FUNCTION F_Leerfahren : BOOL
VAR_INPUT
END_VAR
VAR
END_VAR

(* Netzwerk: 3 Leerfahren *)

(*
	O "M8.1MagLeerf" M8.1 -- Magazin Leerfahren
	O "M8.2SortLeerf" M8.2 -- Sortierer Leerfahren
	S "M 23.1" M23.1 -- Zylinder sollen IN Leerfahrstellung
*)	
IF VAT.bMagazinLeerfahren OR VAT.bSortiererLeerfahren THEN
	VAT.bZylINLeerFahrt := TRUE; //Zylinder sollen IN Leerfahrstellung
END_IF

(*	
	UN "M8.1MagLeerf" M8.1 -- Magazin Leerfahren
	UN "M8.2SortLeerf" M8.2 -- Sortierer Leerfahren
	U "M 23.1" M23.1 -- Zylinder sollen IN Leerfahrstellung
	R "M 23.1" M23.1 -- Zylinder sollen IN Leerfahrstellung
	S "M 23.2" M23.2 -- Zylinder sollen AUS Leerfahrstellung
*)
IF NOT VAT.bMagazinLeerfahren AND
	NOT VAT.bSortiererLeerfahren AND
	VAT.bZylINLeerFahrt THEN
	
	VAT.bZylINLeerFahrt := FALSE;
	VAT.bZylAUSLeerFahrt := TRUE;
END_IF

(*	
	O "M 23.0" M23.0 -- Takt für Vereinzelung bei Leerfahren
	SPBN kl
*)

IF NOT VAT.bTaktVereinzLeerF THEN
	RETURN;
END_IF

(*	
	U "T 41" T41 -- Takt für Magazin leerfahren
	SPB kl
*)
GVL.tofMagazLeerFahr(IN := FALSE, PT := T#500MS);
IF GVL.tofMagazLeerFahr.Q THEN
	RETURN;
END_IF

(*
	L S5T#500MS
	SA "T 41" T41 -- Takt für Magazin leerfahren
	CLR
	SA "T 41" T41 -- Takt für Magazin leerfahren
	
	UN "M 23.0" M23.0 -- Takt für Vereinzelung bei Leerfahren
	= "M 23.0" M23.0 -- Takt für Vereinzelung bei Leerfahren
*)
GVL.tofMagazLeerFahr(IN := TRUE, PT := T#500MS);
VAT.bTaktVereinzLeerF := NOT VAT.bTaktVereinzLeerF;

(*
kl: BLD 130
*)

END_FUNCTION

(* stored: Version 1.1.0.1, ProductVersion 3.1.4024.3
   POU F_Leerfahren: Id {6b9ade98-69de-4b4e-8046-6d83073b01a0}, SpecialFunc None *)
